// TIA Portal V17 export
// export: Created 2024-09-27T18:53:45.6438138Z, ExportSetting WithDefaults, DisplayName Totally Integrated Automation Portal, DisplayVersion V17, DisplayName TIA Portal Openness, DisplayVersion V17, DisplayName TIA Portal Version Control Interface, DisplayVersion V17, DisplayName STEP 7 Professional, DisplayVersion V17, DisplayName STEP 7 Safety, DisplayVersion V17, DisplayName WinCC Professional, DisplayVersion V17
FUNCTION "WYJSCIA" : Void   // FC2, LAD
{ S7_Optimized_Access := 'TRUE' }
VERSION : 0.1
// stored: AutoNumber true, IsIECCheckEnabled false, SetENOAutomatically false, UDAEnableTagReadback false
BEGIN

REGION Network 1: SAFETY OK
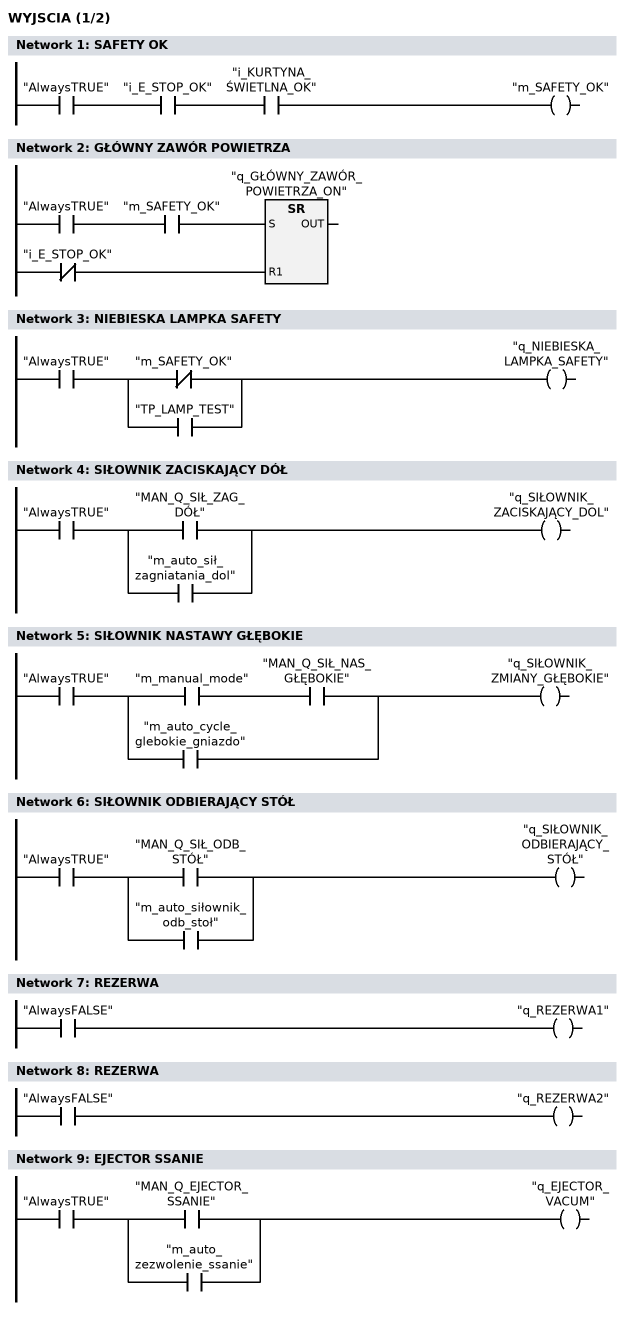
   RUNG wire#powerrail
      Contact( "AlwaysTRUE" )
      Contact( "i_E_STOP_OK" )
      Contact( "i_KURTYNA_ŚWIETLNA_OK" )
      Coil( "m_SAFETY_OK" )
   END_RUNG
   // the same network as SCL:
   "m_SAFETY_OK" := "AlwaysTRUE" AND "i_E_STOP_OK" AND "i_KURTYNA_ŚWIETLNA_OK";
END_REGION

REGION Network 2: GŁÓWNY ZAWÓR POWIETRZA
   RUNG wire#powerrail
      Contact( "AlwaysTRUE" )
      Contact( "m_SAFETY_OK" )
      S_SR(operand := "q_GŁÓWNY_ZAWÓR_POWIETRZA_ON", r1 := wire#w1)
   END_RUNG
   RUNG wire#powerrail
      I_Contact( "i_E_STOP_OK" )
   END_RUNG wire#w1
   // the same network as SCL:
   IF "AlwaysTRUE" AND "m_SAFETY_OK" THEN
       "q_GŁÓWNY_ZAWÓR_POWIETRZA_ON" := TRUE;   // SR flip-flop
   END_IF;
   IF NOT "i_E_STOP_OK" THEN "q_GŁÓWNY_ZAWÓR_POWIETRZA_ON" := FALSE; END_IF;
END_REGION

REGION Network 3: NIEBIESKA LAMPKA SAFETY
   RUNG wire#powerrail
      Contact( "AlwaysTRUE" )
      wire#w1
      I_Contact( "m_SAFETY_OK" )
      wire#w2
      Coil( "q_NIEBIESKA_LAMPKA_SAFETY" )
   END_RUNG
   RUNG wire#w1
      Contact( "TP_LAMP_TEST" )
   END_RUNG wire#w2
   // the same network as SCL:
   "q_NIEBIESKA_LAMPKA_SAFETY" := "AlwaysTRUE" AND (NOT "m_SAFETY_OK" OR "TP_LAMP_TEST");
END_REGION

REGION Network 4: SIŁOWNIK ZACISKAJĄCY DÓŁ
   RUNG wire#powerrail
      Contact( "AlwaysTRUE" )
      wire#w1
      Contact( "MAN_Q_SIŁ_ZAG_DÓŁ" )
      wire#w2
      Coil( "q_SIŁOWNIK_ZACISKAJĄCY_DOL" )
   END_RUNG
   RUNG wire#w1
      Contact( "m_auto_sił_zagniatania_dol" )
   END_RUNG wire#w2
   // the same network as SCL:
   "q_SIŁOWNIK_ZACISKAJĄCY_DOL" := "AlwaysTRUE" AND ("MAN_Q_SIŁ_ZAG_DÓŁ" OR "m_auto_sił_zagniatania_dol");
END_REGION

REGION Network 5: SIŁOWNIK NASTAWY GŁĘBOKIE
   RUNG wire#powerrail
      Contact( "AlwaysTRUE" )
      wire#w1
      Contact( "m_manual_mode" )
      Contact( "MAN_Q_SIŁ_NAS_GŁĘBOKIE" )
      wire#w2
      Coil( "q_SIŁOWNIK_ZMIANY_GŁĘBOKIE" )
   END_RUNG
   RUNG wire#w1
      Contact( "m_auto_cycle_glebokie_gniazdo" )
   END_RUNG wire#w2
   // the same network as SCL:
   "q_SIŁOWNIK_ZMIANY_GŁĘBOKIE" := "AlwaysTRUE" AND (("m_manual_mode" AND "MAN_Q_SIŁ_NAS_GŁĘBOKIE") OR "m_auto_cycle_glebokie_gniazdo");
END_REGION

REGION Network 6: SIŁOWNIK ODBIERAJĄCY STÓŁ
   RUNG wire#powerrail
      Contact( "AlwaysTRUE" )
      wire#w1
      Contact( "MAN_Q_SIŁ_ODB_STÓŁ" )
      wire#w2
      Coil( "q_SIŁOWNIK_ODBIERAJĄCY_STÓŁ" )
   END_RUNG
   RUNG wire#w1
      Contact( "m_auto_siłownik_odb_stoł" )
   END_RUNG wire#w2
   // the same network as SCL:
   "q_SIŁOWNIK_ODBIERAJĄCY_STÓŁ" := "AlwaysTRUE" AND ("MAN_Q_SIŁ_ODB_STÓŁ" OR "m_auto_siłownik_odb_stoł");
END_REGION

REGION Network 7: REZERWA
   RUNG wire#powerrail
      Contact( "AlwaysFALSE" )
      Coil( "q_REZERWA1" )
   END_RUNG
   // the same network as SCL:
   "q_REZERWA1" := "AlwaysFALSE";
END_REGION

REGION Network 8: REZERWA
   RUNG wire#powerrail
      Contact( "AlwaysFALSE" )
      Coil( "q_REZERWA2" )
   END_RUNG
   // the same network as SCL:
   "q_REZERWA2" := "AlwaysFALSE";
END_REGION

REGION Network 9: EJECTOR SSANIE
   RUNG wire#powerrail
      Contact( "AlwaysTRUE" )
      wire#w1
      Contact( "MAN_Q_EJECTOR_SSANIE" )
      wire#w2
      Coil( "q_EJECTOR_VACUM" )
   END_RUNG
   RUNG wire#w1
      Contact( "m_auto_zezwolenie_ssanie" )
   END_RUNG wire#w2
   // the same network as SCL:
   "q_EJECTOR_VACUM" := "AlwaysTRUE" AND ("MAN_Q_EJECTOR_SSANIE" OR "m_auto_zezwolenie_ssanie");
END_REGION

REGION Network 10: EJECTOR PRZEDMUCH
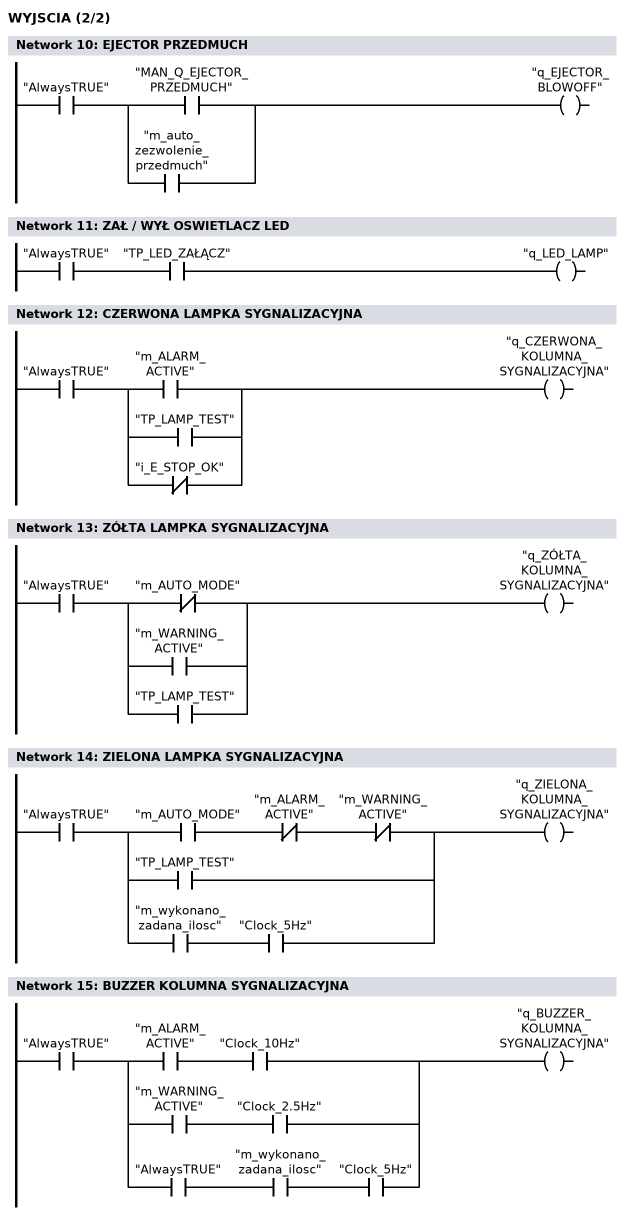
   RUNG wire#powerrail
      Contact( "AlwaysTRUE" )
      wire#w1
      Contact( "MAN_Q_EJECTOR_PRZEDMUCH" )
      wire#w2
      Coil( "q_EJECTOR_BLOWOFF" )
   END_RUNG
   RUNG wire#w1
      Contact( "m_auto_zezwolenie_przedmuch" )
   END_RUNG wire#w2
   // the same network as SCL:
   "q_EJECTOR_BLOWOFF" := "AlwaysTRUE" AND ("MAN_Q_EJECTOR_PRZEDMUCH" OR "m_auto_zezwolenie_przedmuch");
END_REGION

REGION Network 11: ZAŁ / WYŁ OSWIETLACZ LED
   RUNG wire#powerrail
      Contact( "AlwaysTRUE" )
      Contact( "TP_LED_ZAŁĄCZ" )
      Coil( "q_LED_LAMP" )
   END_RUNG
   // the same network as SCL:
   "q_LED_LAMP" := "AlwaysTRUE" AND "TP_LED_ZAŁĄCZ";
END_REGION

REGION Network 12: CZERWONA LAMPKA SYGNALIZACYJNA
   RUNG wire#powerrail
      Contact( "AlwaysTRUE" )
      wire#w1
      Contact( "m_ALARM_ACTIVE" )
      wire#w2
      Coil( "q_CZERWONA_KOLUMNA_SYGNALIZACYJNA" )
   END_RUNG
   RUNG wire#w1
      Contact( "TP_LAMP_TEST" )
   END_RUNG wire#w2
   RUNG wire#w1
      I_Contact( "i_E_STOP_OK" )
   END_RUNG wire#w2
   // the same network as SCL:
   "q_CZERWONA_KOLUMNA_SYGNALIZACYJNA" := "AlwaysTRUE" AND ("m_ALARM_ACTIVE" OR "TP_LAMP_TEST" OR NOT "i_E_STOP_OK");
END_REGION

REGION Network 13: ZÓŁTA LAMPKA SYGNALIZACYJNA
   RUNG wire#powerrail
      Contact( "AlwaysTRUE" )
      wire#w1
      I_Contact( "m_AUTO_MODE" )
      wire#w2
      Coil( "q_ZÓŁTA_KOLUMNA_SYGNALIZACYJNA" )
   END_RUNG
   RUNG wire#w1
      Contact( "m_WARNING_ACTIVE" )
   END_RUNG wire#w2
   RUNG wire#w1
      Contact( "TP_LAMP_TEST" )
   END_RUNG wire#w2
   // the same network as SCL:
   "q_ZÓŁTA_KOLUMNA_SYGNALIZACYJNA" := "AlwaysTRUE" AND (NOT "m_AUTO_MODE" OR "m_WARNING_ACTIVE" OR "TP_LAMP_TEST");
END_REGION

REGION Network 14: ZIELONA LAMPKA SYGNALIZACYJNA
   RUNG wire#powerrail
      Contact( "AlwaysTRUE" )
      wire#w1
      Contact( "m_AUTO_MODE" )
      I_Contact( "m_ALARM_ACTIVE" )
      I_Contact( "m_WARNING_ACTIVE" )
      wire#w2
      Coil( "q_ZIELONA_KOLUMNA_SYGNALIZACYJNA" )
   END_RUNG
   RUNG wire#w1
      Contact( "TP_LAMP_TEST" )
   END_RUNG wire#w2
   RUNG wire#w1
      Contact( "m_wykonano_zadana_ilosc" )
      Contact( "Clock_5Hz" )
   END_RUNG wire#w2
   // the same network as SCL:
   "q_ZIELONA_KOLUMNA_SYGNALIZACYJNA" := "AlwaysTRUE" AND (("m_AUTO_MODE" AND NOT "m_ALARM_ACTIVE" AND NOT "m_WARNING_ACTIVE") OR "TP_LAMP_TEST" OR ("m_wykonano_zadana_ilosc" AND "Clock_5Hz"));
END_REGION

REGION Network 15: BUZZER KOLUMNA SYGNALIZACYJNA
   RUNG wire#powerrail
      Contact( "AlwaysTRUE" )
      wire#w1
      Contact( "m_ALARM_ACTIVE" )
      Contact( "Clock_10Hz" )
      wire#w2
      Coil( "q_BUZZER_KOLUMNA_SYGNALIZACYJNA" )
   END_RUNG
   RUNG wire#w1
      Contact( "m_WARNING_ACTIVE" )
      Contact( "Clock_2.5Hz" )
   END_RUNG wire#w2
   RUNG wire#w1
      Contact( "AlwaysTRUE" )
      Contact( "m_wykonano_zadana_ilosc" )
      Contact( "Clock_5Hz" )
   END_RUNG wire#w2
   // the same network as SCL:
   "q_BUZZER_KOLUMNA_SYGNALIZACYJNA" := "AlwaysTRUE" AND (("m_ALARM_ACTIVE" AND "Clock_10Hz") OR ("m_WARNING_ACTIVE" AND "Clock_2.5Hz") OR ("AlwaysTRUE" AND "m_wykonano_zadana_ilosc" AND "Clock_5Hz"));
END_REGION
END_FUNCTION
